FUNCTION_BLOCK BirthdayManager_1
VAR
	current_date:DATE:=D#2021-7-27;
	person:ARRAY[1..10]OF	T_person:=[(name:='Ali',age:=30,birthday:=D#2020-7-27),
										(name:='Ali',age:=30,birthday:=D#2020-7-27),
										(name:='Ali',age:=30,birthday:=D#2020-7-27),
										(name:='Azmi',age:=36,birthday:=D#2021-7-27),
										(name:='Ali',age:=30,birthday:=D#2020-7-27)];
	i: INT;
	message:string;
	execute: BOOL;
END_VAR

IF	execute	THEN
	FOR i:=1	TO	10	DO
		IF	person[i].birthday=current_date	THEN
			message:='happy Birthday ';
			message:=CONCAT(message,person[i].name);
			person[i].age:=person[i].age+1;
			message:=concat(message,' you are now ');
			message:=concat(message,USINT_TO_STRING(person[i].age));
			execute:=FALSE;
			RETURN;
		END_IF
	END_FOR
END_IF

END_FUNCTION_BLOCK

(* stored: Version 1.1.0.1, ProductVersion 3.1.4024.2
   POU BirthdayManager_1: Id {60f433d5-de24-4da4-a22f-1b47244ffc8b}, SpecialFunc None *)
